FUNCTION Factorial : ULINT
VAR_INPUT
	n: ULINT;
END_VAR
VAR
	nReturnValue: ULINT;
	i: ULINT;
END_VAR

nReturnValue := 1;
FOR i := 1 TO n BY 1 DO
	nReturnValue := nReturnValue * i;
END_FOR
Factorial := nReturnValue;

END_FUNCTION

(* stored: Version 1.1.0.1, ProductVersion 3.1.4024.12
   POU Factorial: Id {3db0ad36-2ec1-474a-81ca-4c1c0cbc1888}, SpecialFunc None *)
